{attribute 'linkalways'} 
{attribute 'no_explicit_call' := 'This FB is a CLASS and must be accessed using methods or properties'}
{attribute 'enable_dynamic_creation'}
FUNCTION_BLOCK Node_F_VN_GetAt_LREAL EXTENDS VisionNode
VAR
    ipContainer : _ITcVnContainer;
    fElement : _LREAL(0.0);
    nIndex : _ULINT(0);
    hrPrev : _HRESULT(S_OK);
    hresult : _HRESULT(S_OK);
END_VAR

METHOD PUBLIC  Clone : I_Node
VAR
	pNode : POINTER TO Node_F_VN_GetAt_LREAL;
END_VAR
pNode := __NEW(Node_F_VN_GetAt_LREAL);
Clone := pNode^;
END_METHOD

METHOD FB_init : BOOL
VAR_INPUT
	bInitRetains : BOOL; // if TRUE, the retain variables are initialized (warm start / cold start)
	bInCopyCode : BOOL;  // if TRUE, the instance afterwards gets moved into the copy code (online change)
END_VAR
AddInput('ipContainer', ipContainer);
AddInput('nIndex', nIndex);
AddInput('hrPrev', hrPrev);
AddOutput('fElement', fElement);
AddOutput('hresult',hresult);
END_METHOD

METHOD PROTECTED OnExecute : HRESULT
hresult.Value := F_VN_GetAt_LREAL(
    ipContainer := ipContainer.Value,
    fElement := fElement.Value,
    nIndex := nIndex.Value,
    hrPrev:= hrPrev.Value);
END_METHOD

METHOD PUBLIC PreExecutionCheck
VAR_INPUT
	Check : I_PreExecutionChecks;
END_VAR
Check.IsTrue(ipContainer.IsValid, 'ipContainer must be a valid container');
Check.IsTrue(ipContainer.HasType(TC_GLOBAL_CONST_LIST.ContainerType_Vector_LREAL), 'ipContainer contains incorrect type');
END_METHOD

END_FUNCTION_BLOCK

(* stored: Version 1.1.0.1, ProductVersion 3.1.4024.13
   POU Node_F_VN_GetAt_LREAL: Id {e75da93c-0f14-4845-9ec1-a99ce8225d3b}, SpecialFunc None
   Folder Constructor: Id {fef6680d-d4a0-49ac-89b4-26a3664e4ee2}
   Method Clone: Id {26a8bc6a-93bc-4ac9-a0ca-e79fc488f32a}
   Method FB_init: Id {d423ad52-799b-442c-83f3-5640ea8ebf91}
   Method OnExecute: Id {442e4bbd-0965-4fde-9658-96bb00754eb2}
   Method PreExecutionCheck: Id {3b24d691-3b6f-4ed9-909a-d61df68d8ef8} *)
